TYPE TcoInsightAcquisitionStatus_v_5_x_x :
STRUCT
    AcquisitionTriggerReady AT %I* : BOOL;
    AcquisitionTriggerAcknowledge AT %I* : BOOL;
    ExposureComplete AT %I* : BOOL;
    MissedAcquisition AT %I* : BOOL;
    OfflineReason0 AT %I* : BOOL;
    OfflineReason1 AT %I* : BOOL;
    OfflineReason2 AT %I* : BOOL;
    Online AT %I* : BOOL;
    AcquisitionID AT %I* : UINT;
END_STRUCT
END_TYPE

(* stored: Version 1.1.0.1, ProductVersion 3.1.4024.11
   DUT TcoInsightAcquisitionStatus_v_5_x_x: Id {326a9b96-4503-0882-004b-7379ed320db0} *)
